Staubli VAL3: Initialisation.pgx

program Initialisation()
begin
  cls()
  resetMotion()
  if bDCY==true
    movej(jDepart,tPince,mRapide)
    userPage()
    put("enter the number of lignes : ")
    get(nLigne)
    taskCreate "Examan_Robot",100,Exam_Robot()
  endIf
end
